# EPICS autosave request: ADPcoWin/iocs/pcocam2IOC/iocBoot/iocPcocam2/auto_settings.req
file "NDStdArrays_settings.req",          P=$(P),  R=image1:
file "commonPlugin_settings.req",         P=$(P)
